Yaskawa INFORM job: R1-WELDTEST.JBI

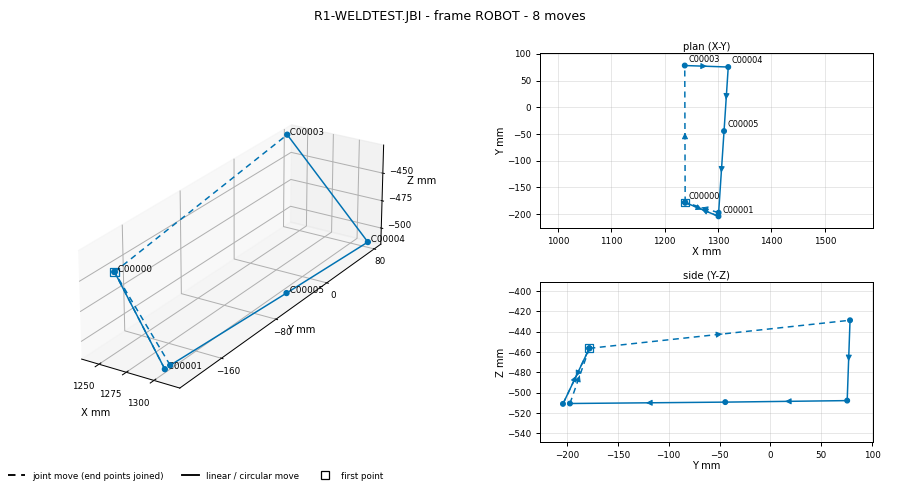
[picture p0: tool path of R1-WELDTEST.JBI in frame ROBOT, 8 of 8 moves have a stored position in this frame; points joined in program order, loops and branches not executed]
/JOB
//NAME R1-WELDTEST
///FOLDERNAME OTHER
//POS
///NPOS 8,8,0,0,0,0
///TOOL 0
///POSTYPE ROBOT
///RECTAN
///RCONF 1,0,1,0,0,0,0,0,0,0,0,0,0,0,0,0,0,0,0,0,0,0,0,0
C00000=1238.525,-178.080,-456.331,22.5427,47.0433,-173.0563
C00001=1300.938,-204.031,-510.994,22.5418,47.0482,-173.0554
C00002=1238.525,-178.080,-456.331,22.5427,47.0433,-173.0563
///RCONF 1,0,1,0,1,0,0,0,0,0,0,0,0,0,0,0,0,0,0,0,0,0,0,0
C00003=1237.753,78.390,-428.724,-11.1636,44.7888,162.3848
C00004=1319.186,75.591,-507.773,-11.1636,44.7888,162.3846
C00005=1311.317,-44.367,-509.259,3.7049,47.6336,173.2330
///RCONF 1,0,1,0,0,0,0,0,0,0,0,0,0,0,0,0,0,0,0,0,0,0,0,0
C00006=1301.172,-197.175,-510.619,18.2801,47.8704,-175.9503
C00007=1238.525,-178.080,-456.331,22.5427,47.0433,-173.0563
///RCONF 0,0,0,0,0,0,0,0,0,0,0,0,0,0,0,0,0,0,0,0,0,0,0,0
BC00000=3683.526
BC00001=3683.520
BC00002=3683.526
BC00003=3683.526
BC00004=3683.526
BC00005=3683.526
BC00006=3683.526
BC00007=3683.526
//INST
///DATE 2024/02/28 12:57
///ATTR SC,RW,RJ
////FRAME ROBOT
///GROUP1 RB1,BS1
NOP
'Tac weld
MACRO1 MJ#(0) ARGF1
MOVJ C00000 BC00000 VJ=10.00
MOVL C00001 BC00001 V=33.3
ARCON
TIMER T=0.60
ARCOF
MOVJ C00002 BC00002 VJ=10.00
PAUSE
PAUSE
'Weld positions
MOVJ C00003 BC00003 VJ=10.00
MACRO1 MJ#(0) ARGF3
MOVL C00004 BC00004 V=33.3
ARCON
MOVL C00005 BC00005 V=9.2
ARCOF
MACRO1 MJ#(0) ARGF4
ARCON
MOVL C00006 BC00006 V=9.2
ARCOF
MOVJ C00007 BC00007 VJ=10.00
END
